(* CODESYS project Uppgift 10.project

Project tree, tasks and I/O mapping:
  Device : CODESYS Control Win V3, 3S - Smart Software Solutions GmbH, order no. 305021, version 3.5.10.40
    application Application
      libraries: Standard, * (System)
      task MainTask (cyclic, interval t#20ms, priority 1) calls PLC_PRG
      program PLC_PRG [LD]
*)

// Device/Application/PLC_PRG
PROGRAM PLC_PRG
VAR
	// Buttons
	Btn_Green: BOOL;
	Btn_Yellow: BOOL;
	Btn_Red: BOOL;
	
	// Timmers
	RTC_0: RTC;
	
	// TimeValues
	TimmerCounter2: DATE_AND_TIME; // Counting value
	TimmerCounter3: DATE_AND_TIME; // Save value
	TimmerCounter4: DATE_AND_TIME; // 0. Default reset value.
	
	// Latch values
	Latch_return_Value: BOOL;
	
END_VAR
VAR // added by the converter: edge detectors and wires of the graphical bodies
    _w1 : BOOL;
END_VAR

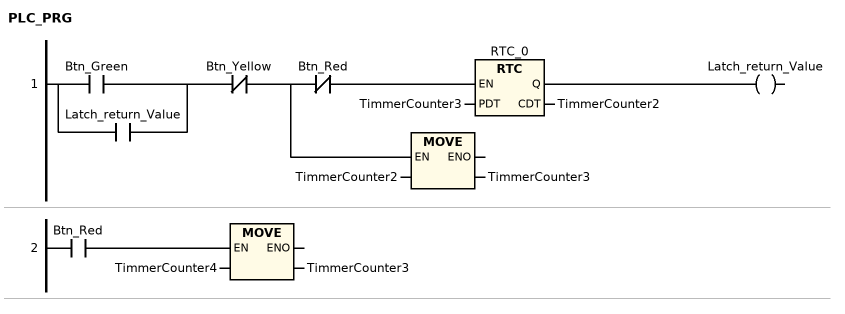
// NETWORK 1
_w1 := (Btn_Green OR Latch_return_Value) AND NOT Btn_Yellow;
RTC_0(EN := _w1 AND NOT Btn_Red, PDT := TimmerCounter3, CDT => TimmerCounter2); // RTC
Latch_return_Value := RTC_0.Q;
IF _w1 THEN TimmerCounter3 := TimmerCounter2; END_IF

// NETWORK 2
IF Btn_Red THEN TimmerCounter3 := TimmerCounter4; END_IF

END_PROGRAM
